// TwinCAT 3 PLC project PLC
// ProjectVersion: 1.0.0
// ProgramVersion: 3.1.4024.0
// libraries:
//   Tc2_Standard, * (Beckhoff Automation GmbH)
//   Tc2_System, * (Beckhoff Automation GmbH)
//   Tc3_EventLogger, * (Beckhoff Automation GmbH)
//   Tc3_JsonXml, * (Beckhoff Automation GmbH)
//   Tc3_Module, * (Beckhoff Automation GmbH)
// project tree:
//   DUTs/ DUT_DriveData_HMI.TcDUT, DUT_ServoRecipe.TcDUT, ST_Alarm.TcDUT, ST_Cylinder.TcDUT, ST_Parent.TcDUT
//   GVLs/ GVL.TcGVL
//   / PlcTask.TcTTO
//   POUs/ MAIN.TcPOU
// real-time tasks:
//   TASK PlcTask: cycle T#10ms, priority 20, ADS port 350

CONFIGURATION PLC
    RESOURCE PLC ON TwinCAT3
        TASK PlcTask(INTERVAL := T#10ms, PRIORITY := 20);
        PROGRAM MAIN WITH PlcTask : MAIN;
    END_RESOURCE
END_CONFIGURATION

// ---- DUTs/DUT_DriveData_HMI.TcDUT
TYPE DUT_DriveData_HMI :
STRUCT
	iHMI_Signal				: INT;
	iMotorSpeed_RPM			: INT;
	rMotorCurrent_Amps		: REAL;
	rMotorTorque_Pcnt		: REAL;
	strDriveError			: STRING(50);
	wDriveFaultCode			: WORD;
	xDriveCommsOk			: BOOL;
	xDriveFault				: BOOL;
	xDriveModeJog			: BOOL;
	xDriveRunning			: BOOL;
	xDriveStopped			: BOOL;
	xDriveAtReference		: BOOL;
	xPB_Jog					: BOOL;
	xPB_Reset				: BOOL;
	xInExecute				: BOOL;
	xInManualControlMode	: BOOL;
	xHasManualRunCommand	: BOOL;
	xManualOpSpeedSelected	: BOOL;
	xManualJogSpeedSelected : BOOL;
	rSpeedSetpointOp_Ips	: REFERENCE TO REAL;
	rSpeedSetpointJog_Ips	: REFERENCE TO REAL;	
END_STRUCT
END_TYPE

// ---- DUTs/DUT_ServoRecipe.TcDUT
TYPE DUT_ServoRecipe :
STRUCT
	LoadPosition			: LREAL;
	GraspPosition			: LREAL;
	PartNumber				: STRING;
	Velocity				: LREAL;
//These were moved here to provide values per part number even though they are not servo parameters
	ClampLeverMaxForceLimit	: LREAL;
	CutTriggerMaxForceLimit : LREAL;
END_STRUCT
END_TYPE

// ---- DUTs/ST_Alarm.TcDUT
TYPE ST_Alarm :
STRUCT
	dtDateTime		: DATE_AND_TIME;
	sName			: STRING;
	nCategory		: DINT;
	nCode			: DINT;
	sMessage		: STRING(255);
END_STRUCT
END_TYPE

// ---- DUTs/ST_Cylinder.TcDUT
TYPE ST_Cylinder :
STRUCT
	ExtendedCmd		: BOOL;
	RetractCmd		: BOOL;
	Extended		: BOOL;
END_STRUCT
END_TYPE

// ---- DUTs/ST_Parent.TcDUT
TYPE ST_Parent :
STRUCT
	stInner		: DUT_ServoRecipe;
	iMember		: DINT;
END_STRUCT
END_TYPE

// ---- GVLs/GVL.TcGVL
{attribute 'qualified_only'}
VAR_GLOBAL
	stTest			: ST_Parent;
	arrCylinders	: ARRAY[0..9] OF ST_Cylinder;
	arrAlarms		: ARRAY[0..31] OF ST_Alarm;
	
	DriveData1		: DUT_DriveData_HMI;
	DriveData2		: DUT_DriveData_HMI;
END_VAR

// ---- POUs/MAIN.TcPOU
PROGRAM MAIN
VAR
	rand	: ARRAY [0..9] OF DRAND;
	ton		: ARRAY [0..9] OF TON;
	fTrend	AT %Q* : ARRAY[0..9] OF LREAL;
	i		: DINT;
	
	iTest1	AT %Q* : DINT;
	iTest2	AT %Q* : DINT;
	
	fbJson			: FB_JsonSaxPrettyWriter;
	fbJsonDataType 	: FB_JsonReadWriteDataType;
	sSer			: STRING(511);
	iJsonLen		: UDINT;
	bRead			: BOOL;
	bWrite			: BOOL;
	
	//fbFileIo		: FB_FileIO;
	
	bInit			: BOOL := TRUE;
	bRaiseAlarm		: BOOL;
	bClear			: BOOL;
	fbFirstAlarm	: FB_TcMessage;
	fbSecondAlarm	: FB_TcAlarm;
END_VAR

IF bInit THEN
	fbSecondAlarm.CreateEx(TC_EVENTS.Alarms.MyFirstAlarm, FALSE, 0);
	bInit := FALSE;
END_IF

IF bRaiseAlarm THEN
	fbSecondAlarm.ipArguments.AddDInt(1001);
	fbSecondAlarm.Raise(0);
	bRaiseAlarm := FALSE;
END_IF

IF bClear THEN
	fbSecondAlarm.Clear(0, TRUE);
	bClear := FALSE;
END_IF

(*
FOR i := 0 TO 9 DO
	rand[i](Seed:=TO_INT(i));
	ton[i](IN:=(NOT ton[i].Q), PT:=TO_TIME(i * 1000));
	
	IF ton[i].Q THEN
		fTrend[i] := rand[i].Num * 10;
	END_IF
END_FOR

IF bRead THEN
	IF fbFileIo.ReadAllText('/test.json', sSer) THEN
		fbJsonDataType.SetSymbolFromJson(sSer, 'DUT_ServoRecipe', SIZEOF(GVL.stTest.stInner), ADR(GVL.stTest.stInner));
		bRead := FALSE;
	END_IF
	//sSer := fbJsonDataType.GetJsonStringFromSymbol('DUT_ServoRecipe' ,SIZEOF(GVL.stTest.stInner), ADR(GVL.stTest.stInner));
	//MEMSET(ADR(GVL.stTest.stInner), 0, SIZEOF(GVL.stTest.stInner)); 
	//bRead := FALSE;
END_IF

IF bWrite THEN
	fbJson.ResetDocument();
	fbJsonDataType.AddJsonValueFromSymbol(fbJson, 'DUT_ServoRecipe', SIZEOF(DUT_ServoRecipe), ADR(GVL.stTest.stInner));
	fbJson.CopyDocument(sSer, SIZEOF(sSer));
	//sSer := fbJsonDataType.GetJsonStringFromSymbol('DUT_ServoRecipe' ,SIZEOF(GVL.stTest.stInner), ADR(GVL.stTest.stInner));
	IF fbFileIo.WriteAllText('/test.json', sSer) THEN
		sSer := '';
		bWrite := FALSE;
	END_IF
END_IF
*)

END_PROGRAM
